FUNCTION_BLOCK NormallyClosedSensor
VAR
	input AT %I*	:	BOOL;
END_VAR

PROPERTY PUBLIC IsActive : BOOL

// ho eliminato manualmente il Setter di questa proprietà perché qui non ha senso
GET
IsActive := NOT input;
END_GET
END_PROPERTY

END_FUNCTION_BLOCK

(* stored: Version 1.1.0.1, ProductVersion 3.1.4024.11
   POU NormallyClosedSensor: Id {cf35b91c-883d-4722-9eb1-85c6733e2d78}, SpecialFunc None
   Property IsActive: Id {bea70df2-ff2b-4195-9ca3-a948b46cb6c4}
   Get Get: Id {e19861bc-5910-46c1-bf54-05096819507a} *)
